(* IEC 61131-3 sources: Lasal/CPU_5344_V01/Class/MotorParaBase, 1 file *)

(* ---- MotorParaBase.st ---- *)
(*!
<Class
	Name               = "MotorParaBase"
	Revision           = "0.0"
	RealtimeTask       = "false"
	CyclicTask         = "false"
	BackgroundTask     = "true"
	DefBackground      = "100 ms"
	Sigmatek           = "false"
	OSInterface        = "false"
	HighPriority       = "false"
	Automatic          = "false"
	UpdateMode         = "Prescan"
	SharedCommandTable = "true"
	Objectsize         = "(480,780)">
	<Channels>
		<Server Name="ClassSvr" Visualized="true" Initialize="false" WriteProtected="false" Retentive="SRam"/>
		<Server Name="FeedbOfffset" Visualized="true" Initialize="false" WriteProtected="false" Retentive="SRam"/>
		<Server Name="P_KV" Visualized="true" Initialize="false" WriteProtected="false" Retentive="SRam"/>
		<Server Name="P_SFF" Visualized="true" Initialize="false" WriteProtected="false" Retentive="SRam"/>
		<Server Name="P_SSCALE" Visualized="true" Initialize="false" WriteProtected="false" Retentive="SRam"/>
		<Server Name="P_TFF" Visualized="true" Initialize="false" WriteProtected="false" Retentive="SRam"/>
		<Server Name="Update" Visualized="false" Initialize="false" WriteProtected="false" Retentive="false"/>
		<Server Name="V_KP" Visualized="true" Initialize="false" WriteProtected="false" Retentive="SRam"/>
		<Server Name="V_KPREL" Visualized="true" Initialize="false" WriteProtected="false" Retentive="SRam"/>
		<Server Name="V_NMAX" Visualized="true" Initialize="false" WriteProtected="false" Retentive="SRam"/>
		<Server Name="V_T" Visualized="true" Initialize="false" WriteProtected="false" Retentive="SRam"/>
		<Server Name="V_T2" Visualized="true" Initialize="false" WriteProtected="false" Retentive="SRam"/>
		<Server Name="V_TN" Visualized="true" Initialize="false" WriteProtected="false" Retentive="SRam"/>
		<Client Name="MotPara" Required="true" Internal="false"/>
		<Client Name="PositionPara" Required="true" Internal="false"/>
		<Client Name="SpeedPara" Required="true" Internal="false"/>
	</Channels>
</Class>
*)
MotorParaBase : CLASS
  //Servers:
	ClassSvr 	: SvrChCmd_DINT;
	Update 	: SvrCh_DINT;
	P_KV 	: SvrCh_DINT;
	P_SFF 	: SvrCh_DINT;
	P_TFF 	: SvrCh_DINT;
	P_SSCALE 	: SvrCh_DINT;
	V_KP 	: SvrCh_DINT;
	V_T 	: SvrCh_DINT;
	V_TN 	: SvrCh_DINT;
	V_T2 	: SvrCh_DINT;
	V_NMAX 	: SvrCh_DINT;
	V_KPREL 	: SvrCh_DINT;
	FeedbOfffset 	: SvrCh_DINT;
  //Clients:
	PositionPara 	: CltChCmd__DrivePositionPara;
	SpeedPara 	: CltChCmd__DriveSpeedPara;
	MotPara 	: CltChCmd__DriveMotorPara;
  //Variables:
		dataLoaded 	: DINT;
		tStartTim 	: UDINT;
  //Functions:

	FUNCTION VIRTUAL GLOBAL Init;

	FUNCTION VIRTUAL GLOBAL Background
		VAR_INPUT
			EAX 	: UDINT;
		END_VAR
		VAR_OUTPUT
			state (EAX) 	: UDINT;
		END_VAR;

	FUNCTION GLOBAL LoadWriteVal;

	FUNCTION VIRTUAL GLOBAL Update::Write
		VAR_INPUT
			input (EAX) 	: DINT;
		END_VAR
		VAR_OUTPUT
			result (EAX) 	: DINT;
		END_VAR;

	FUNCTION VIRTUAL GLOBAL P_KV::Write
		VAR_INPUT
			input (EAX) 	: DINT;
		END_VAR
		VAR_OUTPUT
			result (EAX) 	: DINT;
		END_VAR;

	FUNCTION VIRTUAL GLOBAL P_SFF::Write
		VAR_INPUT
			input (EAX) 	: DINT;
		END_VAR
		VAR_OUTPUT
			result (EAX) 	: DINT;
		END_VAR;

	FUNCTION VIRTUAL GLOBAL P_TFF::Write
		VAR_INPUT
			input (EAX) 	: DINT;
		END_VAR
		VAR_OUTPUT
			result (EAX) 	: DINT;
		END_VAR;

	FUNCTION VIRTUAL GLOBAL P_SSCALE::Write
		VAR_INPUT
			input (EAX) 	: DINT;
		END_VAR
		VAR_OUTPUT
			result (EAX) 	: DINT;
		END_VAR;

	FUNCTION VIRTUAL GLOBAL V_KP::Write
		VAR_INPUT
			input (EAX) 	: DINT;
		END_VAR
		VAR_OUTPUT
			result (EAX) 	: DINT;
		END_VAR;

	FUNCTION VIRTUAL GLOBAL V_T::Write
		VAR_INPUT
			input (EAX) 	: DINT;
		END_VAR
		VAR_OUTPUT
			result (EAX) 	: DINT;
		END_VAR;

	FUNCTION VIRTUAL GLOBAL V_TN::Write
		VAR_INPUT
			input (EAX) 	: DINT;
		END_VAR
		VAR_OUTPUT
			result (EAX) 	: DINT;
		END_VAR;

	FUNCTION VIRTUAL GLOBAL V_T2::Write
		VAR_INPUT
			input (EAX) 	: DINT;
		END_VAR
		VAR_OUTPUT
			result (EAX) 	: DINT;
		END_VAR;

	FUNCTION VIRTUAL GLOBAL V_NMAX::Write
		VAR_INPUT
			input (EAX) 	: DINT;
		END_VAR
		VAR_OUTPUT
			result (EAX) 	: DINT;
		END_VAR;

	FUNCTION VIRTUAL GLOBAL V_KPREL::Write
		VAR_INPUT
			input (EAX) 	: DINT;
		END_VAR
		VAR_OUTPUT
			result (EAX) 	: DINT;
		END_VAR;

	FUNCTION VIRTUAL GLOBAL FeedbOfffset::Write
		VAR_INPUT
			input (EAX) 	: DINT;
		END_VAR
		VAR_OUTPUT
			result (EAX) 	: DINT;
		END_VAR;
  //Tables:
	FUNCTION @STD
		VAR_OUTPUT
			ret_code	: CONFSTATES;
		END_VAR;
	FUNCTION GLOBAL TAB @CT_;
END_CLASS;

#pragma usingLtd _DriveMotorPara
#pragma usingLtd _DrivePositionPara
#pragma usingLtd _DriveSpeedPara

FUNCTION VIRTUAL GLOBAL MotorParaBase::Init

END_FUNCTION

FUNCTION VIRTUAL GLOBAL MotorParaBase::Update::Write
	VAR_INPUT
		input (EAX) 	: DINT;
	END_VAR
	VAR_OUTPUT
		result (EAX) 	: DINT;
	END_VAR

	Update := input;
  LoadWriteVal();
	result := Update;

END_FUNCTION

FUNCTION GLOBAL MotorParaBase::LoadWriteVal

  /// position para
  PositionPara.P_KV := PositionPara.P_KV.Read();
  PositionPara.P_SFF := PositionPara.P_SFF.Read();
  PositionPara.P_TFF := PositionPara.P_TFF.Read();
  PositionPara.P_SSCALE := PositionPara.P_SSCALE.Read();

  if P_KV = 0 then
    P_KV := PositionPara.P_KV;
  end_if;
  if P_SFF = 0 then
    P_SFF := PositionPara.P_SFF;
  end_if;
  if P_TFF = 0 then
    P_TFF := PositionPara.P_TFF;
  end_if;
  if P_SSCALE = 0 then
    P_SSCALE := PositionPara.P_SSCALE;
  end_if;

  // kijk waarden o
  SpeedPara.V_KP := SpeedPara.V_KP.Read();
  SpeedPara.V_T := SpeedPara.V_T.Read();
  SpeedPara.V_TN := SpeedPara.V_TN.Read();
  SpeedPara.V_T2 := speedPara.V_T2.Read();
  SpeedPara.V_NMAX := Speedpara.V_NMAX.Read();
  SpeedPara.V_KPREL := SpeedPara.V_KPREL.Read();

  if V_KP = 0 then
    V_KP := SpeedPara.V_KP;
  end_if;
  if V_T = 0 then
    V_T := SpeedPara.V_T.Read();
  end_if;
  if V_TN = 0 then
    V_TN := SpeedPara.V_TN.Read();
  end_if;
   if V_T2 = 0 then
    V_T2 := SpeedPara.V_T2.Read();
  end_if;
  if V_NMAX = 0 then
    V_NMAX := SpeedPara.V_NMAX.Read();
  end_if;
  if V_KPREL = 0 then
    V_KPREL := SpeedPara.V_KPREL.Read();
  end_if;

  // MotorParaBase
  MotPara.M_ROFF := MotPara.M_ROFF.Read();

  if FeedbOfffset = 0 then
    FeedbOfffset := MotPara.M_ROFF.Read();
  end_if;

  // nu schrijf alle variabelen
  // position para
  PositionPara.P_KV.Write(input:=P_KV);
  PositionPara.P_SFF.Write(input:=P_SFF);
  PositionPara.P_TFF.Write(input:=P_TFF);
  PositionPara.P_SSCALE.Write(input:=P_SSCALE);

  // speed para
  SpeedPara.V_KP.Write(input:=V_KP);
  SpeedPara.V_T.Write(input:=V_T);
  SpeedPara.V_TN.Write(input:=V_TN);
  SpeedPara.V_T2.Write(input:=V_T2);
  SpeedPara.V_NMAX.Write(input:=V_NMAX);
  SpeedPara.V_KPREL.Write(input:=V_KPREL);

  // motor
  MotPara.M_ROFF.Write(input:=FeedbOfffset);

  // refresh
  SpeedPara.RefreshAllPara();

END_FUNCTION

FUNCTION VIRTUAL GLOBAL MotorParaBase::Background
	VAR_INPUT
		EAX 	: UDINT;
	END_VAR
	VAR_OUTPUT
		state (EAX) 	: UDINT;
	END_VAR

	state := READY;

END_FUNCTION

FUNCTION VIRTUAL GLOBAL MotorParaBase::V_KP::Write
	VAR_INPUT
		input (EAX) 	: DINT;
	END_VAR
	VAR_OUTPUT
		result (EAX) 	: DINT;
	END_VAR

	V_KP := input;
	result := V_KP;

  LoadWriteVal();

END_FUNCTION

FUNCTION VIRTUAL GLOBAL MotorParaBase::V_TN::Write
	VAR_INPUT
		input (EAX) 	: DINT;
	END_VAR
	VAR_OUTPUT
		result (EAX) 	: DINT;
	END_VAR

	V_TN := input;
	result := V_TN;

  LoadWriteVal();

END_FUNCTION

FUNCTION VIRTUAL GLOBAL MotorParaBase::V_T::Write
	VAR_INPUT
		input (EAX) 	: DINT;
	END_VAR
	VAR_OUTPUT
		result (EAX) 	: DINT;
	END_VAR

	V_T := input;
	result := V_T;

  LoadWriteVal();

END_FUNCTION

FUNCTION VIRTUAL GLOBAL MotorParaBase::V_T2::Write
	VAR_INPUT
		input (EAX) 	: DINT;
	END_VAR
	VAR_OUTPUT
		result (EAX) 	: DINT;
	END_VAR

	V_T2 := input;
	result := V_T2;

  LoadWriteVal();

END_FUNCTION

FUNCTION VIRTUAL GLOBAL MotorParaBase::V_NMAX::Write
	VAR_INPUT
		input (EAX) 	: DINT;
	END_VAR
	VAR_OUTPUT
		result (EAX) 	: DINT;
	END_VAR

	V_NMAX := input;
	result := V_NMAX;

  LoadWriteVal();

END_FUNCTION

FUNCTION VIRTUAL GLOBAL MotorParaBase::V_KPREL::Write
	VAR_INPUT
		input (EAX) 	: DINT;
	END_VAR
	VAR_OUTPUT
		result (EAX) 	: DINT;
	END_VAR

	V_KPREL := input;
	result := V_KPREL;

  LoadWriteVal();

END_FUNCTION

FUNCTION VIRTUAL GLOBAL MotorParaBase::P_KV::Write
	VAR_INPUT
		input (EAX) 	: DINT;
	END_VAR
	VAR_OUTPUT
		result (EAX) 	: DINT;
	END_VAR

	P_KV := input;
	result := P_KV;
  LoadWriteVal();

END_FUNCTION

FUNCTION VIRTUAL GLOBAL MotorParaBase::P_SFF::Write
	VAR_INPUT
		input (EAX) 	: DINT;
	END_VAR
	VAR_OUTPUT
		result (EAX) 	: DINT;
	END_VAR

	P_SFF := input;
	result := P_SFF;
  LoadWriteVal();

END_FUNCTION

FUNCTION VIRTUAL GLOBAL MotorParaBase::P_TFF::Write
	VAR_INPUT
		input (EAX) 	: DINT;
	END_VAR
	VAR_OUTPUT
		result (EAX) 	: DINT;
	END_VAR

	P_TFF := input;
	result := P_TFF;
  LoadWriteVal();

END_FUNCTION

FUNCTION VIRTUAL GLOBAL MotorParaBase::FeedbOfffset::Write
	VAR_INPUT
		input (EAX) 	: DINT;
	END_VAR
	VAR_OUTPUT
		result (EAX) 	: DINT;
	END_VAR

	FeedbOfffset := input;
	result := FeedbOfffset;
  LoadWriteVal();

END_FUNCTION

FUNCTION VIRTUAL GLOBAL MotorParaBase::P_SSCALE::Write
	VAR_INPUT
		input (EAX) 	: DINT;
	END_VAR
	VAR_OUTPUT
		result (EAX) 	: DINT;
	END_VAR

	P_SSCALE := input;
	result := P_SSCALE;
  LoadWriteVal();

END_FUNCTION
